PROGRAM LiqNaReceita
VAR
	iCounter: INT;
END_VAR

//Esse bloco verifica quais liquidos que estão sendo usados na receita, para que não seja possível iniciar a limpeza neles
FOR iCounter := 1 TO 12 DO
		Liquidos.LiqNaReceita[iCounter] := Receta_Activa.SetCircuitosLiq[iCounter].Paso <> 0;
END_FOR

END_PROGRAM

(* stored: Version 1.1.0.1, ProductVersion 3.1.4024.13
   POU LiqNaReceita: Id {a8c5e6a8-585e-4fb6-b20f-abe3bafe6f03}, SpecialFunc None *)
